FUNCTION_BLOCK AnalogMotorDriver
VAR_INPUT
	// Nominally, respect requested command voltage between (-10)-10V, i.e. if rCommandVoltage
	// is 5, then the output on the channel should be 5V. However, we can alternatively 
	// Request voltage in normalized mode, which considers rCommandVoltage as a 
	// normalized signal between (-1)-1. To enable this mode, set the bUseNormalizedScale
	// flag, which is defaulted to false. When normalized signals are used, the user can additionally 
	// specify whether normalized commands map to (-10)-10V, or (-5)-5V; the latter is triggered
	// when bUseHalfScale is set to TRUE. 
	rCommandVoltage : REAL;
	bUseNormalizedScale : BOOL := FALSE;
	bUseHalfScale : BOOL := FALSE; 
END_VAR
VAR_OUTPUT
	nPosAnalogOutput AT %Q* : INT; 
	nNegAnalogOutput AT %Q* : INT; 
	nZeroRefAnalogOutput AT %Q* : INT; 
	bOutputInError : BOOL; 
END_VAR
VAR
	nTEN_VOLT_AMPLITUDE : INT := 32767; 
	nFIVE_VOLT_AMPLITUDE : INT := 16383;
END_VAR

IF NOT bUseNormalizedScale THEN 
	
	// In this case we were passed a raw voltage signal. 
	// Should check to see if scaling is appropriate, etc. 
	IF ABS(rCommandVoltage) > 10 THEN
		bOutputInError := TRUE; 
		RETURN; 
	END_IF
	
	nPosAnalogOutput := REAL_TO_INT(rCommandVoltage * nTEN_VOLT_AMPLITUDE / 10.0);
	nNegAnalogOutput := -1 * nPosAnalogOutput;  
	bOutputInError := FALSE;

ELSE 
	
	// Again check if argument is valid
	IF ABS(rCommandVoltage) > 1 THEN 
		bOutputInError := TRUE; 
		RETURN;
	END_IF
	
	// Check to see if we should use the half scale. 
	IF bUseHalfScale THEN
		nPosAnalogOutput := REAL_TO_INT(rCommandVoltage * nFIVE_VOLT_AMPLITUDE); 
	ELSE
		nPosAnalogOutput := REAL_TO_INT(rCommandVoltage * nTEN_VOLT_AMPLITUDE); 
	END_IF
	
	nNegAnalogOutput := -1 * nPosAnalogOutput;  
	bOutputInError := FALSE; 
	
END_IF

END_FUNCTION_BLOCK

(* stored: Version 1.1.0.1, ProductVersion 3.1.4024.12
   POU AnalogMotorDriver: Id {b2eb26c5-5ea8-480c-816a-aba06acf678d}, SpecialFunc None *)
